{attribute 'linkalways'} 
{attribute 'no_explicit_call' := 'This FB is a CLASS and must be accessed using methods or properties'}
{attribute 'enable_dynamic_creation'}
FUNCTION_BLOCK Node_F_VN_AddToContainerElements_TcVnVector2_INT EXTENDS VisionNode
VAR
    aValue : _TcVnVector2_INT;
    ipContainer : _ITcVnContainer;
    hrPrev : _HRESULT(S_OK);
    hresult : _HRESULT(S_OK);
END_VAR

METHOD PUBLIC  Clone : I_Node
VAR
    pNode : POINTER TO Node_F_VN_AddToContainerElements_TcVnVector2_INT;
END_VAR
pNode := __NEW(Node_F_VN_AddToContainerElements_TcVnVector2_INT);
Clone := pNode^;
END_METHOD

METHOD FB_init : BOOL
VAR_INPUT
    bInitRetains : BOOL; // if TRUE, the retain variables are initialized (warm start / cold start)
    bInCopyCode : BOOL;  // if TRUE, the instance afterwards gets moved into the copy code (online change)
END_VAR
AddInput('aValue', aValue);
AddInput('ipContainer', ipContainer);
AddInput('hrPrev', hrPrev);
AddOutput('ipContainer', ipContainer);
AddOutput('hresult',hresult);
END_METHOD

METHOD PROTECTED OnExecute
hresult.Value := F_VN_AddToContainerElements_TcVnVector2_INT(
    aValue := aValue.Value,
    ipContainer := ipContainer.Value,
    hrPrev:= hrPrev.Value);
END_METHOD

METHOD PUBLIC PreExecutionCheck
VAR_INPUT
    Check : I_PreExecutionChecks;
END_VAR
Check.IsTrue(ipContainer.IsValid, 'ipContainer must be a valid container');
Check.IsTrue(ipContainer.IsType(TC_GLOBAL_CONST_LIST.ContainerType_Vector_TcVnVector2_INT), 'ipContainer contains incorrect type');
END_METHOD

END_FUNCTION_BLOCK

(* stored: Version 1.1.0.1, ProductVersion 3.1.4026.13
   POU Node_F_VN_AddToContainerElements_TcVnVector2_INT: Id {6615dc52-ec01-4cde-994c-cb6ea6844330}, SpecialFunc None
   Folder Constructor: Id {9e76f4d7-aec2-4014-b8ef-c7d55cfb3593}
   Method Clone: Id {2bb75fe1-6ec0-4eaa-8573-4bfd3c6c44ff}
   Method FB_init: Id {2ed3a265-e98a-4e40-9e58-c9dfcf12e946}
   Method OnExecute: Id {9ef40d3b-fc65-4c41-9fa7-de707329e296}
   Method PreExecutionCheck: Id {697c6ba6-a273-4a61-8d02-9a30aa3c731c} *)
